PROGRAM PRG_Motion


VAR


    END_VAR

END_PROGRAM

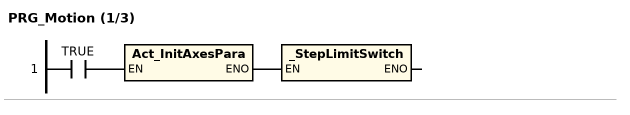
// NETWORK 1
Act_InitAxesPara();
_StepLimitSwitch();

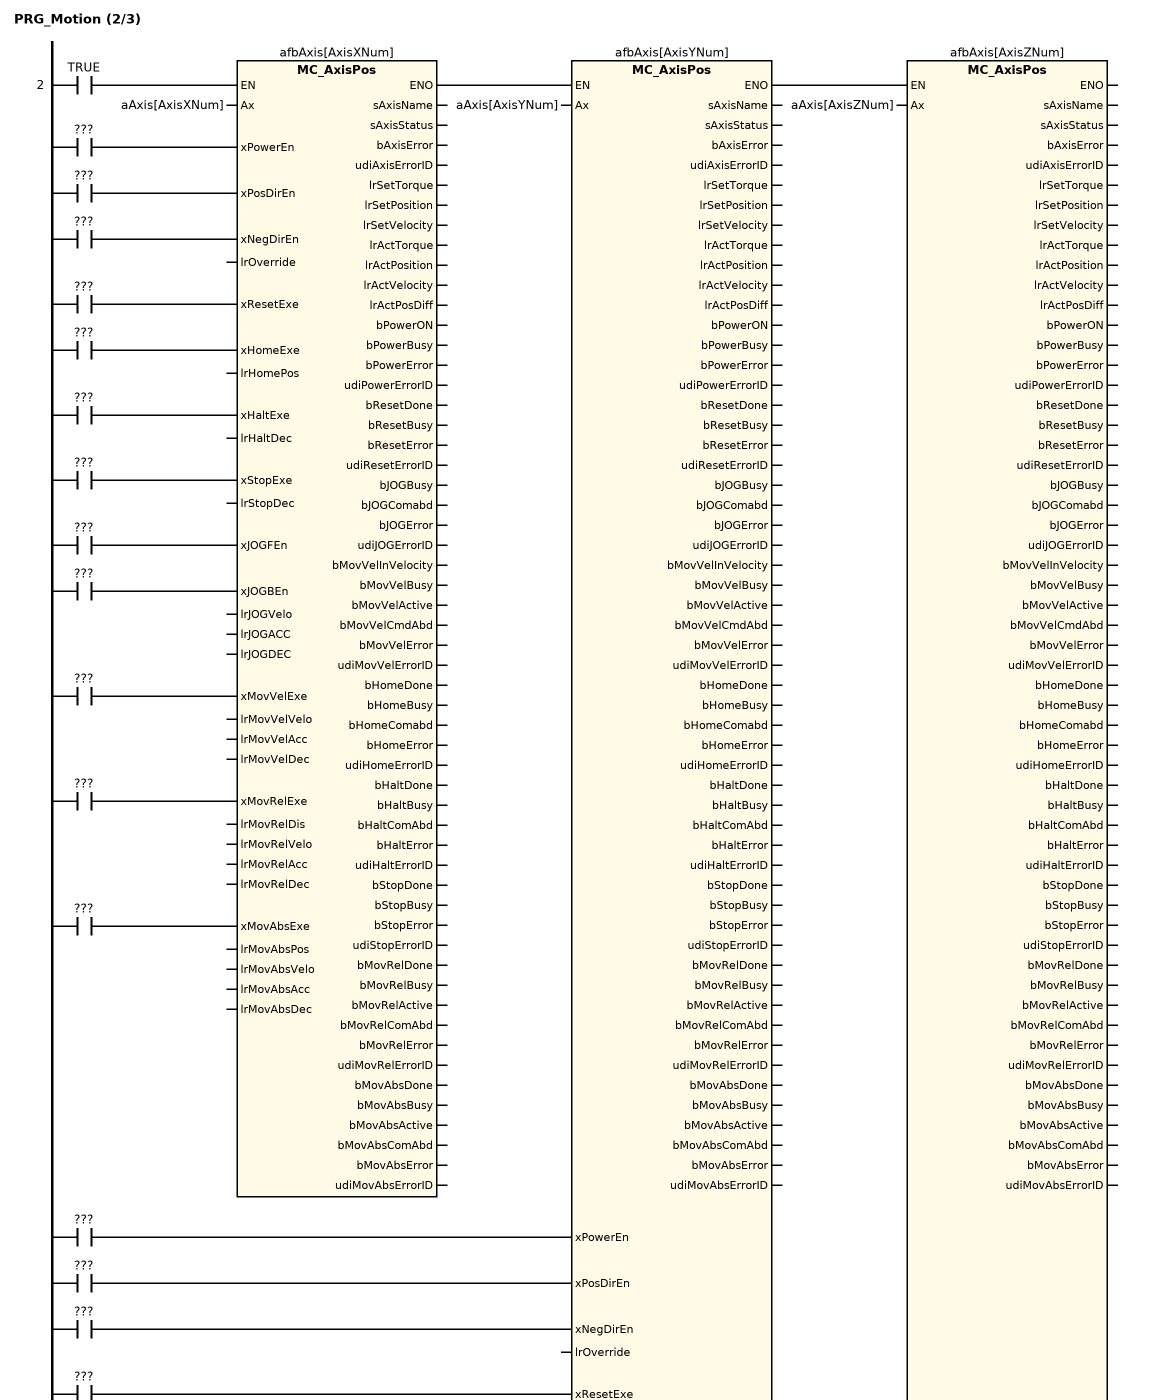
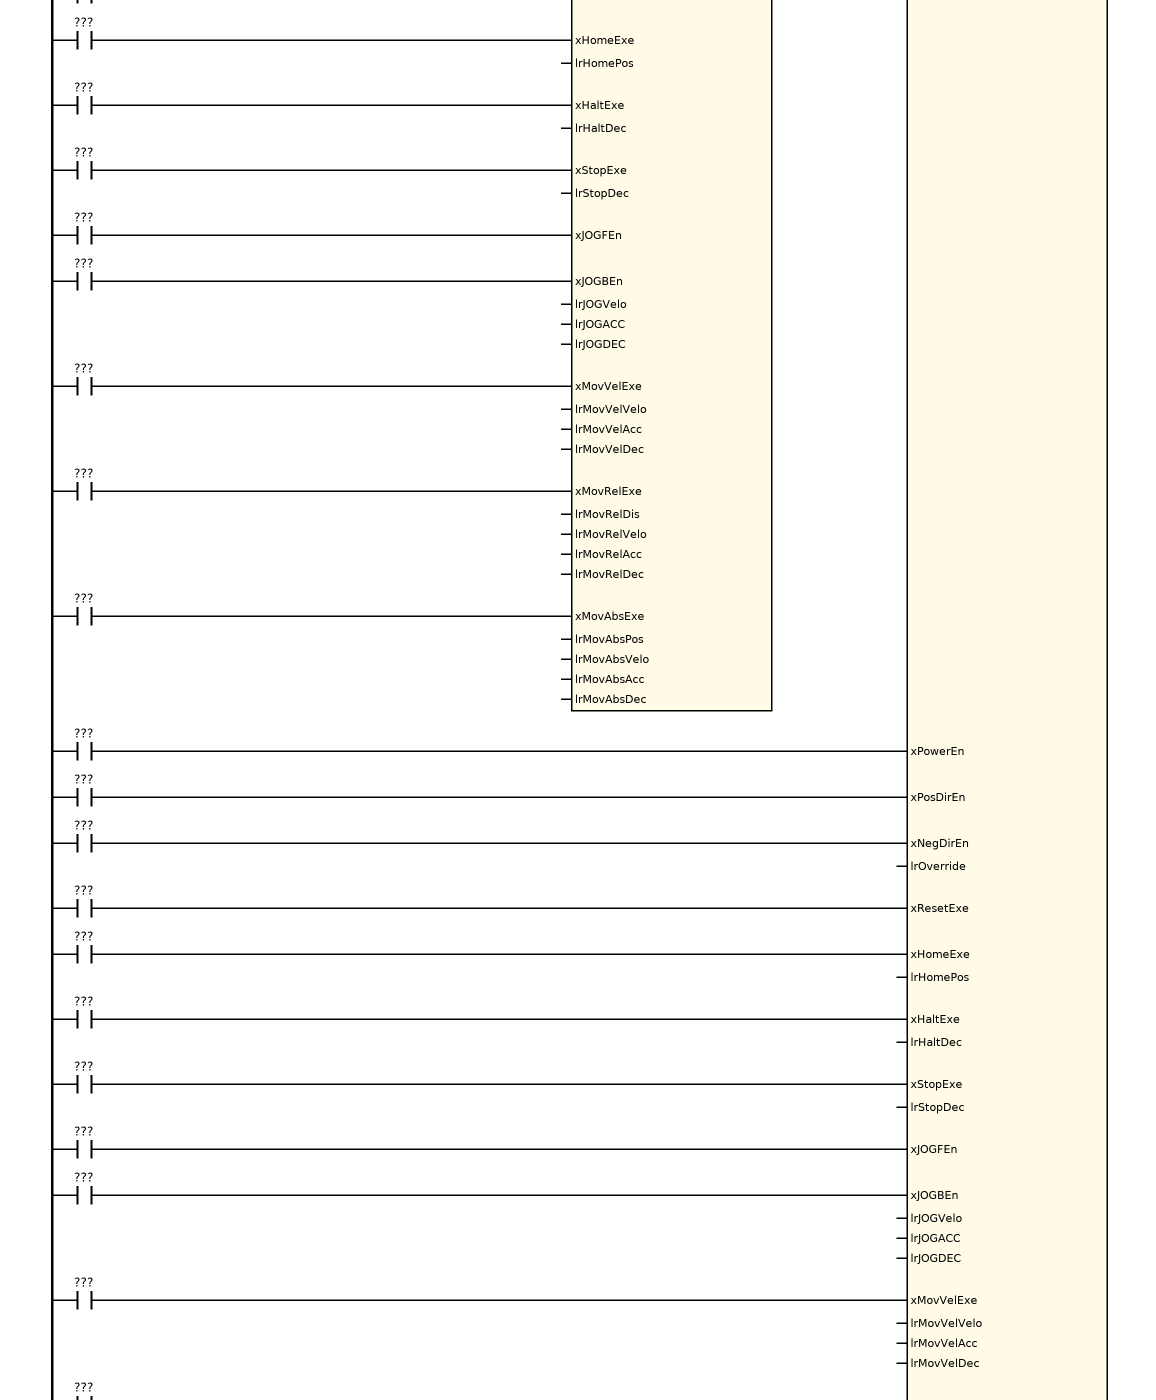
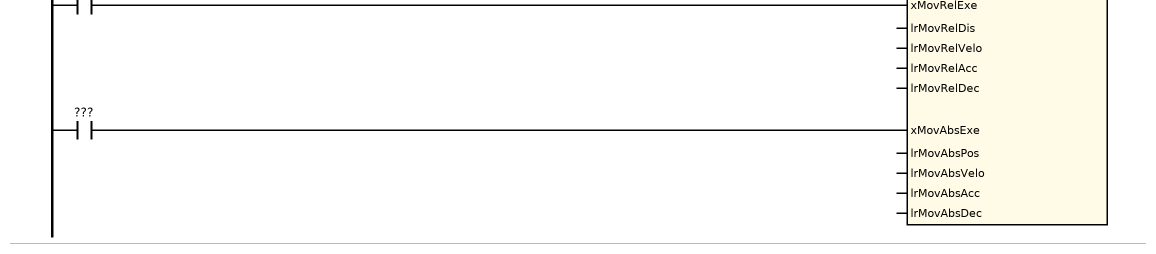
// NETWORK 2
afbAxis[AxisXNum](Ax := aAxis[AxisXNum]); // MC_AxisPos
afbAxis[AxisYNum](Ax := aAxis[AxisYNum]); // MC_AxisPos
afbAxis[AxisZNum](Ax := aAxis[AxisZNum]); // MC_AxisPos

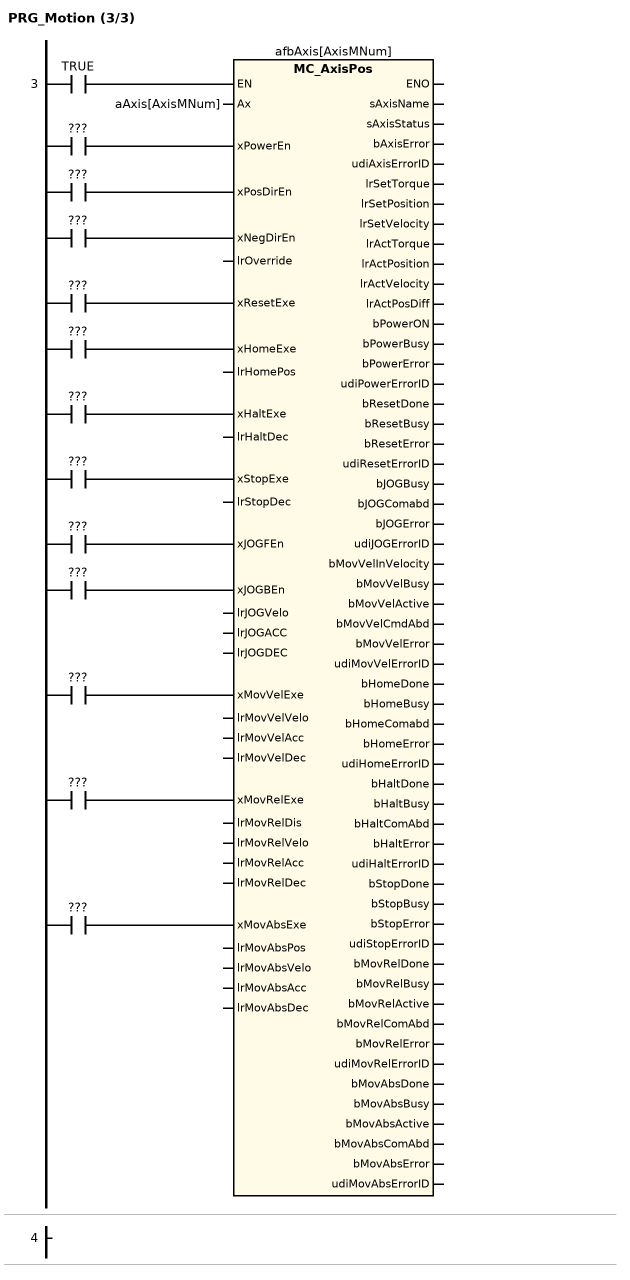
// NETWORK 3
afbAxis[AxisMNum](Ax := aAxis[AxisMNum]); // MC_AxisPos

// NETWORK 4

ACTION _StepLimitSwitch:
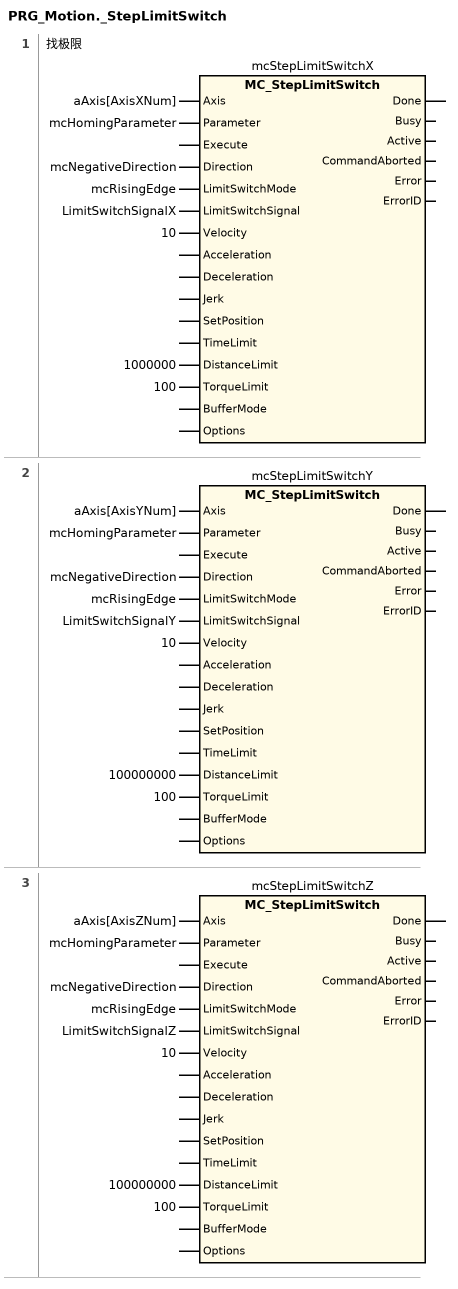
// NETWORK 1: 找极限
mcStepLimitSwitchX(
    Axis := aAxis[AxisXNum],
    Parameter := mcHomingParameter,
    Direction := mcNegativeDirection,
    LimitSwitchMode := mcRisingEdge,
    LimitSwitchSignal := LimitSwitchSignalX,
    Velocity := 10,
    DistanceLimit := 1000000,
    TorqueLimit := 100); // MC_StepLimitSwitch

// NETWORK 2
mcStepLimitSwitchY(
    Axis := aAxis[AxisYNum],
    Parameter := mcHomingParameter,
    Direction := mcNegativeDirection,
    LimitSwitchMode := mcRisingEdge,
    LimitSwitchSignal := LimitSwitchSignalY,
    Velocity := 10,
    DistanceLimit := 100000000,
    TorqueLimit := 100); // MC_StepLimitSwitch

// NETWORK 3
mcStepLimitSwitchZ(
    Axis := aAxis[AxisZNum],
    Parameter := mcHomingParameter,
    Direction := mcNegativeDirection,
    LimitSwitchMode := mcRisingEdge,
    LimitSwitchSignal := LimitSwitchSignalZ,
    Velocity := 10,
    DistanceLimit := 100000000,
    TorqueLimit := 100); // MC_StepLimitSwitch

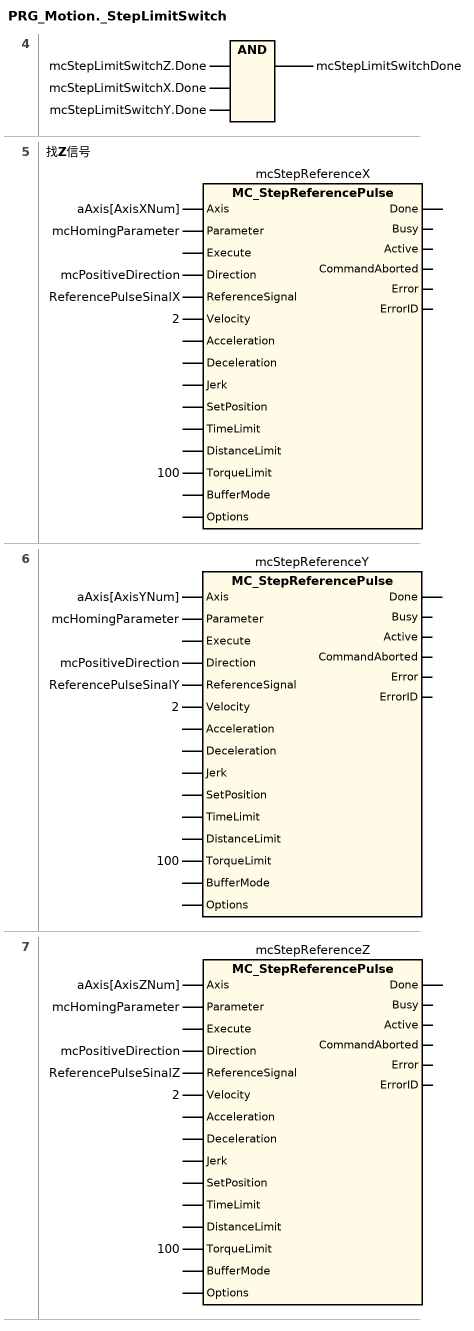
// NETWORK 4
mcStepLimitSwitchDone := mcStepLimitSwitchZ.Done AND mcStepLimitSwitchX.Done AND mcStepLimitSwitchY.Done;

// NETWORK 5: 找Z信号
mcStepReferenceX(
    Axis := aAxis[AxisXNum],
    Parameter := mcHomingParameter,
    Direction := mcPositiveDirection,
    ReferenceSignal := ReferencePulseSinalX,
    Velocity := 2,
    TorqueLimit := 100); // MC_StepReferencePulse

// NETWORK 6
mcStepReferenceY(
    Axis := aAxis[AxisYNum],
    Parameter := mcHomingParameter,
    Direction := mcPositiveDirection,
    ReferenceSignal := ReferencePulseSinalY,
    Velocity := 2,
    TorqueLimit := 100); // MC_StepReferencePulse

// NETWORK 7
mcStepReferenceZ(
    Axis := aAxis[AxisZNum],
    Parameter := mcHomingParameter,
    Direction := mcPositiveDirection,
    ReferenceSignal := ReferencePulseSinalZ,
    Velocity := 2,
    TorqueLimit := 100); // MC_StepReferencePulse

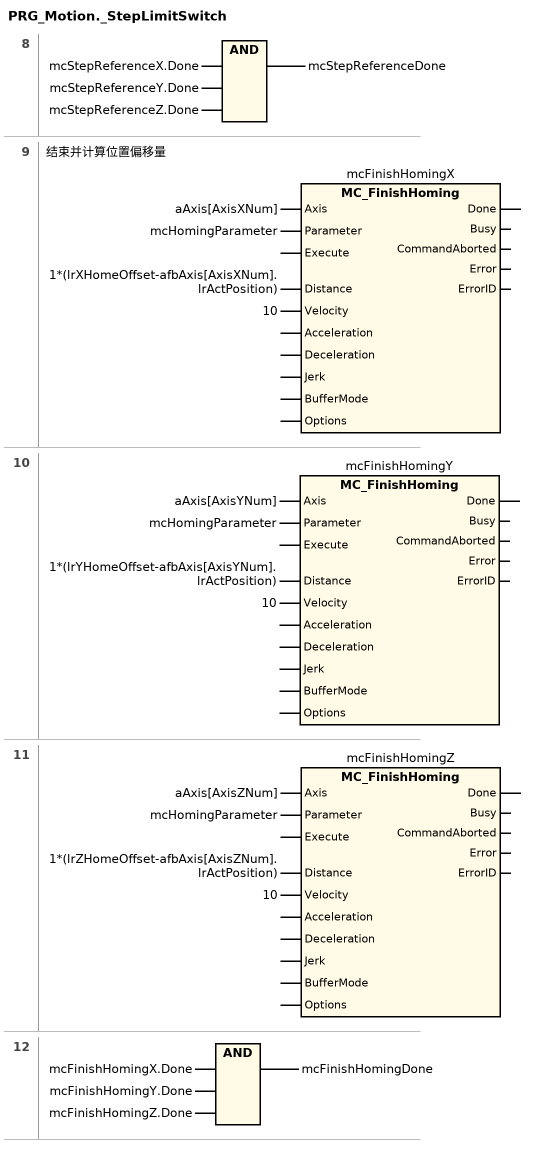
// NETWORK 8
mcStepReferenceDone := mcStepReferenceX.Done AND mcStepReferenceY.Done AND mcStepReferenceZ.Done;

// NETWORK 9: 结束并计算位置偏移量
mcFinishHomingX(
    Axis := aAxis[AxisXNum],
    Parameter := mcHomingParameter,
    Distance := 1*(lrXHomeOffset-afbAxis[AxisXNum].lrActPosition),
    Velocity := 10); // MC_FinishHoming

// NETWORK 10
mcFinishHomingY(
    Axis := aAxis[AxisYNum],
    Parameter := mcHomingParameter,
    Distance := 1*(lrYHomeOffset-afbAxis[AxisYNum].lrActPosition),
    Velocity := 10); // MC_FinishHoming

// NETWORK 11
mcFinishHomingZ(
    Axis := aAxis[AxisZNum],
    Parameter := mcHomingParameter,
    Distance := 1*(lrZHomeOffset-afbAxis[AxisZNum].lrActPosition),
    Velocity := 10); // MC_FinishHoming

// NETWORK 12
mcFinishHomingDone := mcFinishHomingX.Done AND mcFinishHomingY.Done AND mcFinishHomingZ.Done;

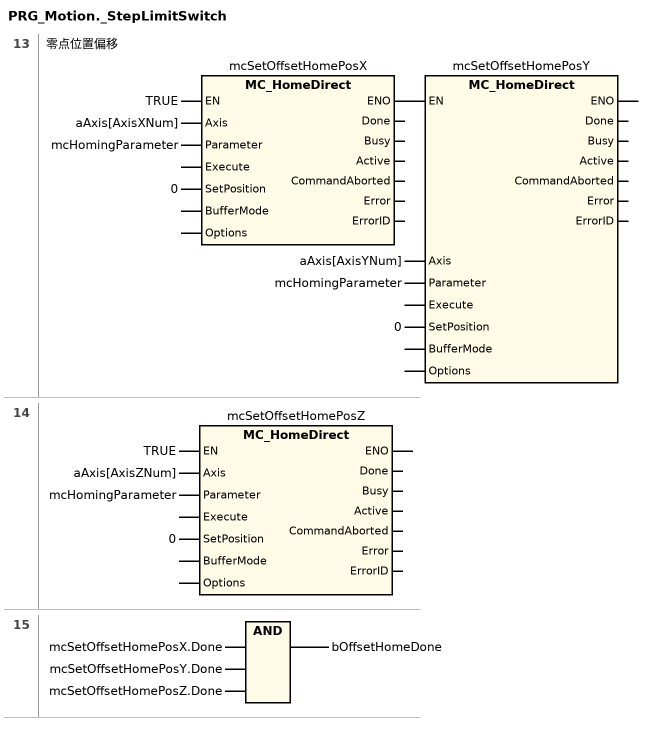
// NETWORK 13: 零点位置偏移
mcSetOffsetHomePosX(Axis := aAxis[AxisXNum], Parameter := mcHomingParameter, SetPosition := 0); // MC_HomeDirect
mcSetOffsetHomePosY(Axis := aAxis[AxisYNum], Parameter := mcHomingParameter, SetPosition := 0); // MC_HomeDirect

// NETWORK 14
mcSetOffsetHomePosZ(Axis := aAxis[AxisZNum], Parameter := mcHomingParameter, SetPosition := 0); // MC_HomeDirect

// NETWORK 15
bOffsetHomeDone := mcSetOffsetHomePosX.Done AND mcSetOffsetHomePosY.Done AND mcSetOffsetHomePosZ.Done;
END_ACTION

ACTION Act_InitAxesPara:
END_PROGRAM

    // 接近开关信号输入与配置


 LimitSwitchSignalX.Level := NOT gIO.bNlimitX;

LimitSwitchSignalY.Level := NOT gIO.bNlimitY;

LimitSwitchSignalZ.Level := NOT gIO.bNlimitZ;


ReferencePulseSinalX.TouchProbe := E_TouchProbe.TouchProbe1;

ReferencePulseSinalX.SignalSource := E_SignalSource.SignalSource_ZeroPulse;


ReferencePulseSinalY.TouchProbe := E_TouchProbe.TouchProbe1;

ReferencePulseSinalY.SignalSource := E_SignalSource.SignalSource_ZeroPulse;


ReferencePulseSinalZ.TouchProbe := E_TouchProbe.TouchProbe1;

ReferencePulseSinalZ.SignalSource := E_SignalSource.SignalSource_ZeroPulse;


    // 第三方驱动器需置真


 mcStepReferenceX.Options.DisableDriveAccess := TRUE;

mcStepReferenceY.Options.DisableDriveAccess := TRUE;

mcStepReferenceZ.Options.DisableDriveAccess := TRUE;

mcFinishHomingX.Options.DisableDriveAccess := TRUE;

mcFinishHomingY.Options.DisableDriveAccess := TRUE;

mcFinishHomingZ.Options.DisableDriveAccess := TRUE;

mcStepLimitSwitchX.Options.DisableDriveAccess := TRUE;

mcStepLimitSwitchY.Options.DisableDriveAccess := TRUE;

mcStepLimitSwitchZ.Options.DisableDriveAccess := TRUE;
END_ACTION

END_PROGRAM

(* stored: Version 1.1.0.1, ProductVersion 3.1.4024.13
   POU PRG_Motion: Id {84960b46-dd7d-4105-99eb-1a63c0803b11}, SpecialFunc None
   Action _StepLimitSwitch: Id {8bce6142-4273-4014-bf70-53d1397d120b}
   Action Act_InitAxesPara: Id {e62f35d6-50be-49cb-a624-18050d4ecb0c} *)
